Staubli VAL3: GetArcAngle.pgx

public program GetArcAngle(trsf x_trTCent, trsf x_trX, trsf x_trY, num& x_nAngle, bool& x_bRes)
  local num l_nDia
  local num l_nLength
  local trsf l_trCenter
  local trsf l_trSource[3]
begin

  l_trSource[0]=x_trTCent
  l_trSource[1]=x_trX
  l_trSource[2]=x_trY


    call Circumcircle(l_trSource,l_trCenter,l_nDia,x_bRes)
  if !x_bRes or l_nDia<=0
    x_bRes=false
    return
  endIf

  l_nLength=distance(l_trSource[0],l_trSource[2])

  if l_nLength>=l_nDia

    x_nAngle=180
  else
      x_nAngle=asin(l_nLength/l_nDia)
  endIf





end
